FUNCTION_BLOCK ListForwardEnumerator_TestSuite EXTENDS TcUnit.FB_TestSuite
VAR
END_VAR

CheckIsValidAtStart();
CheckMoveNextReturnsFalseAtTheEnd();
CheckMoveNextReturnsTrueSingleItem();
CheckMoveNextReturnsFalseWhenEmpty();
CheckMoveNextReturnsTrueMultipleItems();
CheckReset();
CheckTryGet();
CheckTryGetTo();
CheckWorksWithArrays();
CheckWorksWithIntegers();
CheckWorksWithStrings();

METHOD PRIVATE CheckIsValidAtStart
VAR
	result : BOOL;
	enumerator : I_ForwardEnumerator;
END_VAR
VAR_INST
	store : List;
END_VAR
TEST('CheckIsValidAtStart');

enumerator := store.GetEnumerator();

result := enumerator.IsValid;
enumerator.Dispose();

AssertTrue(
	Condition := result,
	Message := 'IsValid returned false'
);

TEST_FINISHED();
END_METHOD

METHOD PRIVATE CheckMoveNextReturnsFalseAtTheEnd
VAR
	in1 : INT := 123;
	result : BOOL;
	enumerator : I_ForwardEnumerator;
END_VAR
VAR_INST
	store : List;
END_VAR
TEST('CheckMoveNextReturnsFalseAtTheEnd');

store.AddItem(in1);
enumerator := store.GetEnumerator();

enumerator.MoveNext();
result := enumerator.MoveNext();
enumerator.Dispose();

AssertFalse(result,
    'MoveNext did not correctly signal the end of the enumeration');
	
TEST_FINISHED();
END_METHOD

METHOD PRIVATE CheckMoveNextReturnsFalseWhenEmpty
VAR
	result : BOOL;
	enumerator : I_ForwardEnumerator;
	count : DINT;
END_VAR
VAR_INST
	store : List;
END_VAR
TEST('CheckMoveNextReturnsFalseWhenEmpty');

count := store.Count;
enumerator := store.GetEnumerator();

result := enumerator.MoveNext();
enumerator.Dispose();

AssertFalse(Condition := result,
    Message := 'MoveNext did not correctly signal the end of the enumeration');

TEST_FINISHED();
END_METHOD

METHOD PRIVATE CheckMoveNextReturnsTrueMultipleItems
VAR
	in1 : INT := 123;
	in2 : INT := 456;
	in3 : INT := 789;
	result : BOOL;
	enumerator : I_ForwardEnumerator;
END_VAR
VAR_INST
	store : List;
END_VAR
TEST('CheckMoveNextReturnsTrueMultipleItems');

store.AddItem(in1);
store.AddItem(in2);
store.AddItem(in3);
enumerator := store.GetEnumerator();

result := enumerator.MoveNext();
enumerator.Dispose();

AssertTrue(result, 'MoveNext did not correctly signal there were more items to follow');

TEST_FINISHED();
END_METHOD

METHOD PRIVATE CheckMoveNextReturnsTrueSingleItem
VAR
	in1 : INT := 123;
	result : BOOL;
	enumerator : I_ForwardEnumerator;
END_VAR
VAR_INST
	store : List;
END_VAR
TEST('CheckMoveNextReturnsTrueSingleItem');

store.AddItem(in1);
enumerator := store.GetEnumerator();

result := enumerator.MoveNext();
enumerator.Dispose();

AssertTrue(result,
    'MoveNext did not correctly signal there were more items to follow');
	
TEST_FINISHED();
END_METHOD

METHOD PRIVATE CheckReset
VAR
	in1 : ARRAY [0..1] OF REAL := [0.1,2.3];
	in2 : ARRAY [0..1] OF REAL := [1.2,3.4];
	in3 : ARRAY [0..1] OF REAL := [2.3,4.5];
	out : ARRAY [0..1] OF REAL;
	expected : ARRAY [0..1] OF REAL := [0.1,2.3];
	enumerator : I_ForwardEnumerator;
END_VAR
VAR_INST
	store : List;
END_VAR
TEST('CheckReset');

store.AddItem(in1);
store.AddItem(in2);
store.AddItem(in3);

enumerator := store.GetEnumerator();

enumerator.MoveNext();
enumerator.MoveNext();
enumerator.Reset();
enumerator.MoveNext();
enumerator.TryGet(out);

enumerator.Dispose();

AssertEquals(
	Expected := expected,
	Actual := out,
	Message := 'Did not produce the expected result'
);

TEST_FINISHED();
END_METHOD

METHOD PRIVATE CheckTryGet
VAR
	in : INT := 123;
	out : INT;
	expected : INT := 123;
	result : BOOL;
	enumerator : I_ForwardEnumerator;
END_VAR
VAR_INST
	store : List;
END_VAR
TEST('CheckTryGet');

store.AddItem(in);
enumerator := store.GetEnumerator();
enumerator.MoveNext();

result := enumerator.TryGet(out);
enumerator.Dispose();

AssertTrue(
	Condition := result,
	Message := 'Method returned false'
);

AssertEquals(
	Expected := expected,
	Actual := out,
	Message := 'Did not produce the expected result'
);

TEST_FINISHED();
END_METHOD

METHOD PRIVATE CheckTryGetTo
VAR
	in : INT := 123;
	out : INT;
	expected : INT := 123;
	result : BOOL;
	enumerator : I_ForwardEnumerator;
END_VAR
VAR_INST
	store : List;
END_VAR
TEST('CheckTryGetTo');

store.AddItem(in);
enumerator := store.GetEnumerator();
enumerator.MoveNext();

result := enumerator.TryGetTo(ADR(out),SIZEOF(out));
enumerator.Dispose();

AssertTrue(
	Condition := result,
	Message := 'Method returned false'
);

AssertEquals(
	Expected := expected,
	Actual := out,
	Message := 'Did not produce the expected result'
);

TEST_FINISHED();
END_METHOD

METHOD PRIVATE CheckWorksWithArrays
VAR
	in1 : ARRAY [0..1] OF REAL := [0.1,2.3];
	in2 : ARRAY [0..1] OF REAL := [1.2,3.4];
	in3 : ARRAY [0..1] OF REAL := [2.3,4.5];
	out1 : ARRAY [0..1] OF REAL;
	out2 : ARRAY [0..1] OF REAL;
	out3 : ARRAY [0..1] OF REAL;
	expected1 : ARRAY [0..1] OF REAL := [0.1,2.3];
	expected2 : ARRAY [0..1] OF REAL := [1.2,3.4];
	expected3 : ARRAY [0..1] OF REAL := [2.3,4.5];
	enumerator : I_ForwardEnumerator;
END_VAR
VAR_INST
	store : List;
END_VAR
TEST('CheckWorksWithArrays');

store.AddItem(in1);
store.AddItem(in2);
store.AddItem(in3);

enumerator := store.GetEnumerator();

enumerator.MoveNext();
enumerator.TryGet(out1);
enumerator.MoveNext();
enumerator.TryGet(out2);
enumerator.MoveNext();
enumerator.TryGet(out3);

enumerator.Dispose();

AssertEquals(
	Expected := expected1,
	Actual := out1,
	Message := 'Did not produce the expected 1st result'
);

AssertEquals(
	Expected := expected2,
	Actual := out2,
	Message := 'Did not produce the expected 2nd result'
);

AssertEquals(
	Expected := expected3,
	Actual := out3,
	Message := 'Did not produce the expected 3rd result'
);

TEST_FINISHED();
END_METHOD

METHOD PRIVATE CheckWorksWithIntegers
VAR
	in1 : INT := 123;
	in2 : INT := 234;
	in3 : INT := 345;
	out1 : INT;
	out2 : INT;
	out3 : INT;
	expected1 : INT := 123;
	expected2 : INT := 234;
	expected3 : INT := 345;
	enumerator : I_ForwardEnumerator;
END_VAR
VAR_INST
	store : List;
END_VAR
TEST('CheckWorksWithIntegers');

store.AddItem(in1);
store.AddItem(in2);
store.AddItem(in3);

enumerator := store.GetEnumerator();

enumerator.MoveNext();
enumerator.TryGet(out1);
enumerator.MoveNext();
enumerator.TryGet(out2);
enumerator.MoveNext();
enumerator.TryGet(out3);

enumerator.Dispose();

AssertEquals(
	Expected := expected1,
	Actual := out1,
	Message := 'Did not produce the expected 1st result'
);

AssertEquals(
	Expected := expected2,
	Actual := out2,
	Message := 'Did not produce the expected 2nd result'
);

AssertEquals(
	Expected := expected3,
	Actual := out3,
	Message := 'Did not produce the expected 3rd result'
);

TEST_FINISHED();
END_METHOD

METHOD PRIVATE CheckWorksWithStrings
VAR
	in1 : STRING := 'test1';
	in2 : STRING := 'test2';
	in3 : STRING := 'test3';
	out1 : STRING;
	out2 : STRING;
	out3 : STRING;
	expected1 : STRING := 'test1';
	expected2 : STRING := 'test2';
	expected3 : STRING := 'test3';
	enumerator : I_ForwardEnumerator;
END_VAR
VAR_INST
	store : List;
END_VAR
TEST('CheckWorksWithStrings');

store.AddItem(in1);
store.AddItem(in2);
store.AddItem(in3);

enumerator := store.GetEnumerator();

enumerator.MoveNext();
enumerator.TryGet(out1);
enumerator.MoveNext();
enumerator.TryGet(out2);
enumerator.MoveNext();
enumerator.TryGet(out3);

enumerator.Dispose();

AssertEquals(
	Expected := expected1,
	Actual := out1,
	Message := 'Did not produce the expected 1st result'
);

AssertEquals(
	Expected := expected2,
	Actual := out2,
	Message := 'Did not produce the expected 2nd result'
);

AssertEquals(
	Expected := expected3,
	Actual := out3,
	Message := 'Did not produce the expected 3rd result'
);

TEST_FINISHED();
END_METHOD

END_FUNCTION_BLOCK

(* stored: Version 1.1.0.1, ProductVersion 3.1.4026.6
   POU ListForwardEnumerator_TestSuite: Id {71bc6d90-25f6-4e5f-ab81-b2ed2832edc4}, SpecialFunc None
   Method CheckIsValidAtStart: Id {78ec5459-0471-41e4-9478-97cb099386b3}
   Method CheckMoveNextReturnsFalseAtTheEnd: Id {57822c53-79e9-48d2-8700-1c3954dbf639}
   Method CheckMoveNextReturnsFalseWhenEmpty: Id {e9136119-78de-43d2-84ab-945aef56b7f7}
   Method CheckMoveNextReturnsTrueMultipleItems: Id {9fc63489-8671-4879-8c50-9441e0fc20e6}
   Method CheckMoveNextReturnsTrueSingleItem: Id {9afc510e-415a-4767-9031-a424bf95bfff}
   Method CheckReset: Id {b6502110-0631-48e1-8f8a-7ca9cd139b28}
   Method CheckTryGet: Id {f2f76693-e8cc-4d6d-9a29-2238540f129c}
   Method CheckTryGetTo: Id {a10234d2-180c-4de5-ae7a-380f60b3c725}
   Method CheckWorksWithArrays: Id {fc714a4d-38d9-48ac-9c82-e49aaf8d36b5}
   Method CheckWorksWithIntegers: Id {2b00fa39-4eda-42f7-ada4-33e201e5f9c3}
   Method CheckWorksWithStrings: Id {3fea921e-4163-4be1-8520-a34ae51f9b32} *)
